FUNCTION_BLOCK WirelessMove 
VAR_INPUT

	sm : FB_SerialCom_Remote; //SerialRemote Assigned to Gantry
	WindowScaling : INT := 1; //Scaling Factor for target window distance
END_VAR
VAR
	XTar : DINT;
	YTar : DINT;
END_VAR
VAR_IN_OUT
		HookX : EtherCat_Kid;
	HookY : EtherCat_Kid;
END_VAR

IF sm.DeadmanPressed >=1 AND SM.Age < T#800MS THEN
	IF Hookx.currentPosition + (((ABS(sm.xAxis) * sm.xAxis) * WindowScaling) / -50) > -1000000 OR Hookx.currentPosition + (((ABS(sm.xAxis) * sm.xAxis) * WindowScaling) / -50) < 1000000 THEN
		XTar := Hookx.currentPosition + (((ABS(sm.xAxis) * sm.xAxis) * WindowScaling) / -50);
	END_IF
	IF HookY.currentPosition + (((ABS(sm.YAxis) * sm.YAxis) * WindowScaling) / -25) > -1000000 OR HookY.currentPosition + (((ABS(sm.YAxis) * sm.YAxis) * WindowScaling) / -25) < 100000 THEN
			YTar := HookY.currentPosition + (((ABS(sm.YAxis) * sm.YAxis) * WindowScaling) / -25);
	END_IF

	main.XTAR := xtar;
	main.YTar := Ytar;
	Main.Kid[hookX.CheckIn.KidID].TargetPos := XTar;
	Main.Kid[Hooky.CheckIn.KidID].TargetPos := YTar;
	//HookY.TargetPos := YTar;
	ELSE
		Main.Kid[hookX.CheckIn.KidID].TargetPos := Main.Kid[hookX.CheckIn.KidID].Currentposition;
		Main.Kid[Hooky.CheckIn.KidID].TargetPos := Main.Kid[Hooky.CheckIn.KidID].CurrentPosition;

END_IF

END_FUNCTION_BLOCK

(* stored: Version 1.1.0.1, ProductVersion 3.1.4022.3
   POU WirelessMove: Id {b316f284-7991-4299-9f9b-1c26edbfde02}, SpecialFunc None *)
